FUNCTION_BLOCK FB_TestHTTP_Options
VAR_INPUT
	fbClient : REFERENCE TO FB_IotHttpClient;
END_VAR
VAR
	
	fbRequest: FB_IotHttpRequest;
	fbJson: FB_JsonDomParser;
	bSend : BOOL;
	bContinuous : BOOL;
	state : UDINT;
	
	RisingEdge		: R_TRIG;
	
	sJson: STRING(1024);		
	sContent: STRING(1024);
	sAllow: STRING(100);
	
	bJsonRes : BOOL;
	jsonDoc    : SJsonValue;
	jsonVal    : SJsonValue;
		
	reqCount : UDINT;		
	invResCount : UDINT := 0;
	invResValCount : UDINT := 0;
	resVal:STRING;
	nResCnt : UDINT;
	nErrCnt1 : UDINT;
	nErrCnt2 : UDINT;
		
	valOkCount: UDINT;	
	
	sUri: STRING(255) := '/posts';
	eRequestType : ETcIotHttpRequestType := ETcIotHttpRequestType.HTTP_OPTIONS;		
END_VAR

RisingEdge( CLK:= bSend );
CASE state OF
0:	
	IF fbClient.bConfigured AND (RisingEdge.Q OR bContinuous) THEN 
		IF fbRequest.SendRequest(sUri:=sUri, fbClient:=fbClient, eRequestType:=eRequestType, 0, 0, 0) THEN				
			state := 1;
			reqCount:=reqCount+1;
		END_IF					
	END_IF
1:
	IF NOT fbRequest.bBusy THEN
			IF NOT fbRequest.bError THEN
				//IF f Access-Control-Allow-Methods: GET,HEAD,PUT,PATCH,POST,DELETE				 
				//;
				IF fbRequest.GetHeaderField('Access-Control-Allow-Methods', ADR(sAllow), SIZEOF(sAllow)) THEN 
					IF Find(sAllow, 'POST') <> 0 THEN
						valOkCount:=valOkCount+1;
					ELSE
						invResValCount:=invResValCount+1;
					END_IF
				ELSE
					invResCount:=invResCount+1;
				END_IF								
			ELSE
				nErrCnt2:=nErrCnt2+1;
			END_IF
			state :=0;				
	END_IF  	
END_CASE
fbClient.Execute();

END_FUNCTION_BLOCK

(* stored: Version 1.1.0.1, ProductVersion 3.1.4024.0
   POU FB_TestHTTP_Options: Id {672fcbbc-79c8-46d2-84e7-e503c0714184}, SpecialFunc None *)
